{attribute 'hide'}
FUNCTION_BLOCK IsValueEven_Test EXTENDS TcUnit.FB_TestSuite

EvenUSINTReturnsTrue();
EvenUINTReturnsTrue();
EvenUDINTReturnsTrue();
EvenULINTReturnsTrue();
EvenSINTReturnsTrue();
EvenINTReturnsTrue();
EvenDINTReturnsTrue();
EvenLINTReturnsTrue();
OddUSINTReturnsFalse();
OddUINTReturnsFalse();
OddUDINTReturnsFalse();
OddULINTReturnsFalse();
OddSINTReturnsFalse();
OddINTReturnsFalse();
OddDINTReturnsFalse();
OddLINTReturnsFalse();

METHOD EvenDINTReturnsTrue
VAR
	result : BOOL;
	value : DINT;
END_VAR
TEST('EvenDINTReturnsTrue');

// @TEST-FIXTURE
value := DINT#2;

// @TEST-RUN
result := IsValueEven(value);

// @TEST-ASSSERT
AssertTrue(Condition := result,
           Message := 'Even DINT did not return TRUE');

TEST_FINISHED();
END_METHOD

METHOD EvenINTReturnsTrue
VAR
	result : BOOL;
	value : INT;
END_VAR
TEST('EvenINTReturnsTrue');

// @TEST-FIXTURE
value := INT#2;

// @TEST-RUN
result := IsValueEven(value);

// @TEST-ASSSERT
AssertTrue(Condition := result,
           Message := 'Even INT did not return TRUE');

TEST_FINISHED();
END_METHOD

METHOD EvenLINTReturnsTrue
VAR
	result : BOOL;
	value : LINT;
END_VAR
TEST('EvenLINTReturnsTrue');

// @TEST-FIXTURE
value := LINT#2;

// @TEST-RUN
result := IsValueEven(value);

// @TEST-ASSSERT
AssertTrue(Condition := result,
           Message := 'Even LINT did not return TRUE');

TEST_FINISHED();
END_METHOD

METHOD EvenSINTReturnsTrue
VAR
	result : BOOL;
	value : SINT;
END_VAR
TEST('EvenSINTReturnsTrue');

// @TEST-FIXTURE
value := SINT#2;

// @TEST-RUN
result := IsValueEven(value);

// @TEST-ASSSERT
AssertTrue(Condition := result,
           Message := 'Even SINT did not return TRUE');

TEST_FINISHED();
END_METHOD

METHOD EvenUDINTReturnsTrue
VAR
	result : BOOL;
	value : UDINT;
END_VAR
TEST('EvenUDINTReturnsTrue');

// @TEST-FIXTURE
value := UDINT#2;

// @TEST-RUN
result := IsValueEven(value);

// @TEST-ASSSERT
AssertTrue(Condition := result,
           Message := 'Even UDINT did not return TRUE');

TEST_FINISHED();
END_METHOD

METHOD EvenUINTReturnsTrue
VAR
	result : BOOL;
	value : UINT;
END_VAR
TEST('EvenUINTReturnsTrue');

// @TEST-FIXTURE
value := UINT#2;

// @TEST-RUN
result := IsValueEven(value);

// @TEST-ASSSERT
AssertTrue(Condition := result,
           Message := 'Even UINT did not return TRUE');

TEST_FINISHED();
END_METHOD

METHOD EvenULINTReturnsTrue
VAR
	result : BOOL;
	value : ULINT;
END_VAR
TEST('EvenULINTReturnsTrue');

// @TEST-FIXTURE
value := ULINT#2;

// @TEST-RUN
result := IsValueEven(value);

// @TEST-ASSSERT
AssertTrue(Condition := result,
           Message := 'Even ULINT did not return TRUE');

TEST_FINISHED();
END_METHOD

METHOD EvenUSINTReturnsTrue
VAR
	result : BOOL;
	value : USINT;
END_VAR
TEST('EvenUSINTReturnsTrue');

// @TEST-FIXTURE
value := USINT#2;

// @TEST-RUN
result := IsValueEven(value);

// @TEST-ASSSERT
AssertTrue(Condition := result,
           Message := 'Even USINT did not return TRUE');

TEST_FINISHED();
END_METHOD

METHOD OddDINTReturnsFalse
VAR
	result : BOOL;
	value : DINT;
END_VAR
TEST('OddDINTReturnsFalse');

// @TEST-FIXTURE
value := DINT#1;

// @TEST-RUN
result := IsValueEven(value);

// @TEST-ASSSERT
AssertFalse(Condition := result,
           Message := 'Odd DINT did not return FALSE');

TEST_FINISHED();
END_METHOD

METHOD OddINTReturnsFalse
VAR
	result : BOOL;
	value : INT;
END_VAR
TEST('OddINTReturnsFalse');

// @TEST-FIXTURE
value := INT#1;

// @TEST-RUN
result := IsValueEven(value);

// @TEST-ASSSERT
AssertFalse(Condition := result,
           Message := 'Odd INT did not return FALSE');

TEST_FINISHED();
END_METHOD

METHOD OddLINTReturnsFalse
VAR
	result : BOOL;
	value : LINT;
END_VAR
TEST('OddLINTReturnsFalse');

// @TEST-FIXTURE
value := LINT#1;

// @TEST-RUN
result := IsValueEven(value);

// @TEST-ASSSERT
AssertFalse(Condition := result,
           Message := 'Odd LINT did not return FALSE');

TEST_FINISHED();
END_METHOD

METHOD OddSINTReturnsFalse
VAR
	result : BOOL;
	value : SINT;
END_VAR
TEST('OddSINTReturnsFalse');

// @TEST-FIXTURE
value := SINT#1;

// @TEST-RUN
result := IsValueEven(value);

// @TEST-ASSSERT
AssertFalse(Condition := result,
           Message := 'Odd SINT did not return FALSE');

TEST_FINISHED();
END_METHOD

METHOD OddUDINTReturnsFalse
VAR
	result : BOOL;
	value : UDINT;
END_VAR
TEST('OddUDINTReturnsFalse');

// @TEST-FIXTURE
value := UDINT#1;

// @TEST-RUN
result := IsValueEven(value);

// @TEST-ASSSERT
AssertFalse(Condition := result,
           Message := 'Odd UDINT did not return FALSE');

TEST_FINISHED();
END_METHOD

METHOD OddUINTReturnsFalse
VAR
	result : BOOL;
	value : UINT;
END_VAR
TEST('OddUINTReturnsFalse');

// @TEST-FIXTURE
value := UINT#1;

// @TEST-RUN
result := IsValueEven(value);

// @TEST-ASSSERT
AssertFalse(Condition := result,
           Message := 'Odd UINT did not return FALSE');

TEST_FINISHED();
END_METHOD

METHOD OddULINTReturnsFalse
VAR
	result : BOOL;
	value : ULINT;
END_VAR
TEST('OddULINTReturnsFalse');

// @TEST-FIXTURE
value := ULINT#1;

// @TEST-RUN
result := IsValueEven(value);

// @TEST-ASSSERT
AssertFalse(Condition := result,
           Message := 'Odd ULINT did not return FALSE');

TEST_FINISHED();
END_METHOD

METHOD OddUSINTReturnsFalse
VAR
	result : BOOL;
	value : USINT;
END_VAR
TEST('OddUSINTReturnsFalse');

// @TEST-FIXTURE
value := USINT#1;

// @TEST-RUN
result := IsValueEven(value);

// @TEST-ASSSERT
AssertFalse(Condition := result,
           Message := 'Odd USINT did not return FALSE');

TEST_FINISHED();
END_METHOD

END_FUNCTION_BLOCK

(* stored: Version 1.1.0.1, ProductVersion 3.1.4024.9
   POU IsValueEven_Test: Id {2d060640-842e-4cab-96ce-8ccd00836465}, SpecialFunc None
   Method EvenDINTReturnsTrue: Id {9227ff4a-9a21-43fa-b594-99401576c53d}
   Method EvenINTReturnsTrue: Id {6a7d083b-4b34-40e4-a63f-487e7e1dd06f}
   Method EvenLINTReturnsTrue: Id {a12a6861-5689-4889-891d-10746982f281}
   Method EvenSINTReturnsTrue: Id {6589d0fa-657f-4aa9-a67c-896e9699418e}
   Method EvenUDINTReturnsTrue: Id {b9125cbc-8a65-4f3c-8642-211bb1877620}
   Method EvenUINTReturnsTrue: Id {c0fbafea-8ee7-4939-bbfa-795ae07dc9a9}
   Method EvenULINTReturnsTrue: Id {1f688b0b-e5ad-4358-a667-dc0df94cfc22}
   Method EvenUSINTReturnsTrue: Id {e2a67179-c219-470f-a863-1b771aa5cdf2}
   Method OddDINTReturnsFalse: Id {e6ab6e8a-6aeb-42c2-a865-ce5a2d7ce825}
   Method OddINTReturnsFalse: Id {5c3a758e-375e-447d-acbf-5bc707cdc54d}
   Method OddLINTReturnsFalse: Id {bb85558c-9ff4-4aff-b7f4-def1315af1c2}
   Method OddSINTReturnsFalse: Id {fad614b6-3821-427f-8f53-7f7b944004c9}
   Method OddUDINTReturnsFalse: Id {97a67a33-b543-4f8c-81e3-583111370ffc}
   Method OddUINTReturnsFalse: Id {5bb6a7ea-ae99-4898-b863-50f0eb74e8d4}
   Method OddULINTReturnsFalse: Id {09c50642-38c0-4129-aa7a-45b6148a1097}
   Method OddUSINTReturnsFalse: Id {d582b2b5-970a-4d48-a8c1-a22a1c25018e} *)
